FUNCTION_BLOCK FB_ConsumptionCalculator
VAR_INPUT
END_VAR
VAR_OUTPUT
	sum : REAL;
END_VAR
VAR
    running       : BOOL;
    elapsedTime   : TIME;
	RTRIG_Started : R_TRIG;
END_VAR

METHOD calculate : BOOL
VAR_INPUT
	start : BOOL;
	valuePerSec : REAL;
    intervalS : INT;
    dtime : TIME;   
END_VAR
VAR
    intervalTime : TIME;
END_VAR
intervalTime := INT_TO_TIME(intervalS*1000);
RTRIG_Started(CLK := start);
// Start edge
IF RTRIG_Started.q THEN
    running := TRUE;
    sum := 0.0;
    elapsedTime := T#0S;
END_IF

IF NOT start THEN
	running := FALSE;
END_IF

IF running THEN
	// Simulate time passing
	elapsedTime := elapsedTime + dtime;
	IF elapsedTime >= intervalTime THEN
		sum := sum + valuePerSec*(intervalS);
		elapsedTime := T#0S;
	END_IF 	
END_IF
END_METHOD

METHOD reset : BOOL
VAR_INPUT
END_VAR

sum := 0;
running := FALSE;
elapsedTime := T#0S;
END_METHOD

END_FUNCTION_BLOCK

(* stored: Version 1.1.0.1, ProductVersion 3.1.4024.9
   POU FB_ConsumptionCalculator: Id {63cec99f-4d10-42e9-916c-b9d1bf4cf7fa}, SpecialFunc None
   Method calculate: Id {6ec4bf84-1c05-4759-9ccd-9c5136c91915}
   Method reset: Id {3a15dc05-77fa-4e69-99b8-7f8aca08106a} *)
